// TIA Portal project "babu_washingMachine" (V15)

(* hardware
DEVICE "S7-1200 station_1"  S7-1200 Station
   slot 0: "Rack_0"  S7-1200 Rack  Rack  V1.0
   slot 1: "PLC_1"  CPU 1212C DC/DC/DC  6ES7 212-1AE40-0XB0  V4.2
*)

// ===== PLC "PLC_1"  CPU 1212C DC/DC/DC =====

VAR_GLOBAL   // PLC tag table "Default tag table"
   "START PB" AT %M0.5 : Bool;
   "CYCLE_ON" AT %M0.7 : Bool;
   "WATER FILLING" AT %Q0.0 : Bool;
   "AGITATION" AT %Q0.1 : Bool;
   "WATER DRAIN" AT %Q0.3 : Bool;
   "SPINNING" AT %Q0.6 : Bool;
   "ALARAM_" AT %Q1.0 : Bool;
END_VAR

VAR_GLOBAL   // PLC tag table "Tag table_1"
   "PUSH BUTTON" AT %M0.0 : Bool;
   "WATER FILLED" AT %M0.1 : Bool;
   "WATER TAP" AT %Q0.2 : Bool;
   "AGITATION COMPLETED" AT %M0.3 : Bool;
   "PUSH BUTTON USED" AT %M0.2 : Bool;
   "DRAIN TAP" AT %Q0.4 : Bool;
   "DRAIN COMPLETE" AT %M0.4 : Bool;
   "SPINNING MOTOR" AT %Q0.5 : Bool;
   "SPINNING COMPLETE" AT %M0.6 : Bool;
   "ALARM" AT %Q0.7 : Bool;
   "ALARM COMPLETED" AT %M1.0 : Bool;
END_VAR

// folder: System blocks/Program resources

DATA_BLOCK "IEC_Timer_0_DB"   // DB1
{ S7_Optimized_Access := 'TRUE' }
AUTHOR : Simatic
FAMILY : IEC
NAME : IEC_TMR
VERSION : 1.0
// stored: InstanceOfName IEC_TIMER
"IEC_TIMER"
BEGIN
END_DATA_BLOCK

DATA_BLOCK "IEC_Timer_0_DB_1"   // DB2
{ S7_Optimized_Access := 'TRUE' }
AUTHOR : Simatic
FAMILY : IEC
NAME : IEC_TMR
VERSION : 1.0
// stored: InstanceOfName IEC_TIMER
"IEC_TIMER"
BEGIN
END_DATA_BLOCK

DATA_BLOCK "IEC_Timer_0_DB_2"   // DB3
{ S7_Optimized_Access := 'TRUE' }
AUTHOR : Simatic
FAMILY : IEC
NAME : IEC_TMR
VERSION : 1.0
// stored: InstanceOfName IEC_TIMER
"IEC_TIMER"
BEGIN
END_DATA_BLOCK

DATA_BLOCK "IEC_Timer_0_DB_3"   // DB4
{ S7_Optimized_Access := 'TRUE' }
AUTHOR : Simatic
FAMILY : IEC
NAME : IEC_TMR
VERSION : 1.0
// stored: InstanceOfName IEC_TIMER
"IEC_TIMER"
BEGIN
END_DATA_BLOCK

DATA_BLOCK "IEC_Timer_0_DB_4"   // DB5
{ S7_Optimized_Access := 'TRUE' }
AUTHOR : Simatic
FAMILY : IEC
NAME : IEC_TMR
VERSION : 1.0
// stored: InstanceOfName IEC_TIMER
"IEC_TIMER"
BEGIN
END_DATA_BLOCK

DATA_BLOCK "IEC_Timer_0_DB_5"   // DB6
{ S7_Optimized_Access := 'TRUE' }
AUTHOR : Simatic
FAMILY : IEC
NAME : IEC_TMR
VERSION : 1.0
// stored: InstanceOfName IEC_TIMER
"IEC_TIMER"
BEGIN
END_DATA_BLOCK

DATA_BLOCK "IEC_Timer_0_DB_6"   // DB7
{ S7_Optimized_Access := 'TRUE' }
AUTHOR : Simatic
FAMILY : IEC
NAME : IEC_TMR
VERSION : 1.0
// stored: InstanceOfName IEC_TIMER
"IEC_TIMER"
BEGIN
END_DATA_BLOCK

DATA_BLOCK "IEC_Timer_0_DB_7"   // DB8
{ S7_Optimized_Access := 'TRUE' }
AUTHOR : Simatic
FAMILY : IEC
NAME : IEC_TMR
VERSION : 1.0
// stored: InstanceOfName IEC_TIMER
"IEC_TIMER"
BEGIN
END_DATA_BLOCK

DATA_BLOCK "IEC_Timer_0_DB_8"   // DB9
{ S7_Optimized_Access := 'TRUE' }
AUTHOR : Simatic
FAMILY : IEC
NAME : IEC_TMR
VERSION : 1.0
// stored: InstanceOfName IEC_TIMER
"IEC_TIMER"
BEGIN
END_DATA_BLOCK

DATA_BLOCK "IEC_Timer_0_DB_9"   // DB10
{ S7_Optimized_Access := 'TRUE' }
AUTHOR : Simatic
FAMILY : IEC
NAME : IEC_TMR
VERSION : 1.0
// stored: InstanceOfName IEC_TIMER
"IEC_TIMER"
BEGIN
END_DATA_BLOCK

DATA_BLOCK "IEC_Timer_0_DB_10"   // DB11
{ S7_Optimized_Access := 'TRUE' }
AUTHOR : Simatic
FAMILY : IEC
NAME : IEC_TMR
VERSION : 1.0
// stored: InstanceOfName IEC_TIMER
"IEC_TIMER"
BEGIN
END_DATA_BLOCK

DATA_BLOCK "IEC_Timer_0_DB_11"   // DB12
{ S7_Optimized_Access := 'TRUE' }
AUTHOR : Simatic
FAMILY : IEC
NAME : IEC_TMR
VERSION : 1.0
// stored: InstanceOfName IEC_TIMER
"IEC_TIMER"
BEGIN
END_DATA_BLOCK

DATA_BLOCK "IEC_Timer_0_DB_12"   // DB13
{ S7_Optimized_Access := 'TRUE' }
AUTHOR : Simatic
FAMILY : IEC
NAME : IEC_TMR
VERSION : 1.0
// stored: InstanceOfName IEC_TIMER
"IEC_TIMER"
BEGIN
END_DATA_BLOCK

DATA_BLOCK "IEC_Timer_0_DB_13"   // DB14
{ S7_Optimized_Access := 'TRUE' }
AUTHOR : Simatic
FAMILY : IEC
NAME : IEC_TMR
VERSION : 1.0
// stored: InstanceOfName IEC_TIMER
"IEC_TIMER"
BEGIN
END_DATA_BLOCK

// folder: (top level)

ORGANIZATION_BLOCK "Main"   // OB1, LAD, ProgramCycle
TITLE = "Main Program Sweep (Cycle)"
{ S7_Optimized_Access := 'TRUE' }
VERSION : 0.1
   VAR_INPUT
      Initial_Call : Bool;   // Initial call of this OB
      Remanence : Bool;   // =True, if remanent data are available
   END_VAR
   VAR_TEMP   // added for the SCL form of the ladder/FBD networks
      _w1 : Bool;
   END_VAR
BEGIN

REGION Network 1
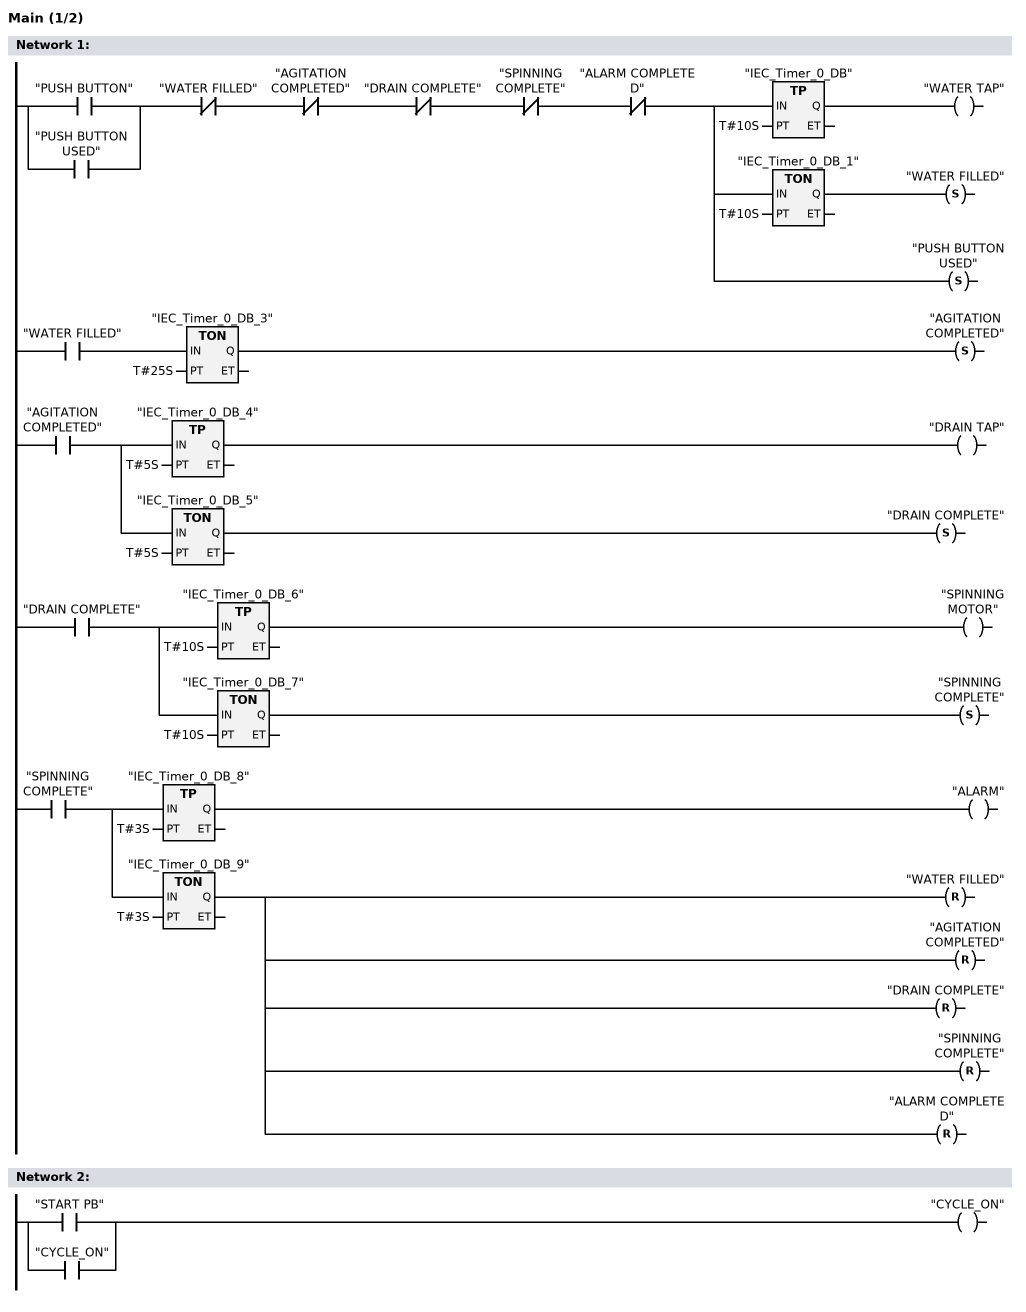
   #_w1 := ("PUSH BUTTON" OR "PUSH BUTTON USED") AND NOT "WATER FILLED" AND NOT "AGITATION COMPLETED" AND NOT "DRAIN COMPLETE" AND NOT "SPINNING COMPLETE" AND NOT "ALARM COMPLETED";
   "IEC_Timer_0_DB".TP(IN := #_w1, PT := T#10S);
   "WATER TAP" := "IEC_Timer_0_DB".Q;
   "IEC_Timer_0_DB_1".TON(IN := #_w1, PT := T#10S);
   IF "IEC_Timer_0_DB_1".Q THEN "WATER FILLED" := TRUE; END_IF;
   IF #_w1 THEN "PUSH BUTTON USED" := TRUE; END_IF;
   "IEC_Timer_0_DB_3".TON(IN := "WATER FILLED", PT := T#25S);
   IF "IEC_Timer_0_DB_3".Q THEN "AGITATION COMPLETED" := TRUE; END_IF;
   "IEC_Timer_0_DB_4".TP(IN := "AGITATION COMPLETED", PT := T#5S);
   "DRAIN TAP" := "IEC_Timer_0_DB_4".Q;
   "IEC_Timer_0_DB_5".TON(IN := "AGITATION COMPLETED", PT := T#5S);
   IF "IEC_Timer_0_DB_5".Q THEN "DRAIN COMPLETE" := TRUE; END_IF;
   "IEC_Timer_0_DB_6".TP(IN := "DRAIN COMPLETE", PT := T#10S);
   "SPINNING MOTOR" := "IEC_Timer_0_DB_6".Q;
   "IEC_Timer_0_DB_7".TON(IN := "DRAIN COMPLETE", PT := T#10S);
   IF "IEC_Timer_0_DB_7".Q THEN "SPINNING COMPLETE" := TRUE; END_IF;
   "IEC_Timer_0_DB_8".TP(IN := "SPINNING COMPLETE", PT := T#3S);
   "ALARM" := "IEC_Timer_0_DB_8".Q;
   "IEC_Timer_0_DB_9".TON(IN := "SPINNING COMPLETE", PT := T#3S);
   IF "IEC_Timer_0_DB_9".Q THEN
       "WATER FILLED" := FALSE;
       "AGITATION COMPLETED" := FALSE;
       "DRAIN COMPLETE" := FALSE;
       "SPINNING COMPLETE" := FALSE;
       "ALARM COMPLETED" := FALSE;
   END_IF;
END_REGION

REGION Network 2
   RUNG wire#powerrail
      Contact( "START PB" )
      wire#w1
      Coil( "CYCLE_ON" )
   END_RUNG
   RUNG wire#powerrail
      Contact( "CYCLE_ON" )
   END_RUNG wire#w1
   // the same network as SCL:
   "CYCLE_ON" := "START PB" OR "CYCLE_ON";
END_REGION

REGION Network 3
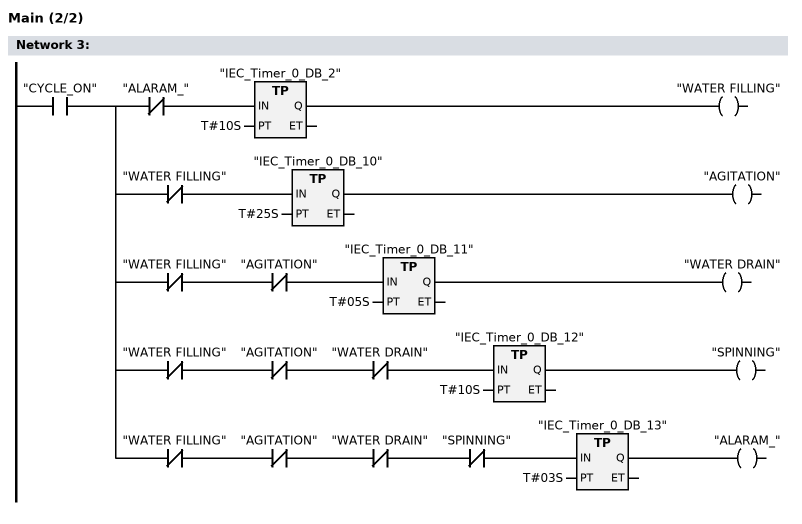
   "IEC_Timer_0_DB_2".TP(IN := "CYCLE_ON" AND NOT "ALARAM_", PT := T#10S);
   "WATER FILLING" := "IEC_Timer_0_DB_2".Q;
   "IEC_Timer_0_DB_10".TP(IN := "CYCLE_ON" AND NOT "WATER FILLING", PT := T#25S);
   "AGITATION" := "IEC_Timer_0_DB_10".Q;
   "IEC_Timer_0_DB_11".TP(IN := "CYCLE_ON" AND NOT "WATER FILLING" AND NOT "AGITATION", PT := T#05S);
   "WATER DRAIN" := "IEC_Timer_0_DB_11".Q;
   "IEC_Timer_0_DB_12".TP(IN := "CYCLE_ON" AND NOT "WATER FILLING" AND NOT "AGITATION" AND NOT "WATER DRAIN",
                          PT := T#10S);
   "SPINNING" := "IEC_Timer_0_DB_12".Q;
   "IEC_Timer_0_DB_13".TP(IN := "CYCLE_ON" AND NOT "WATER FILLING" AND NOT "AGITATION" AND NOT "WATER DRAIN" AND NOT "SPINNING",
                          PT := T#03S);
   "ALARAM_" := "IEC_Timer_0_DB_13".Q;
END_REGION
END_ORGANIZATION_BLOCK